// SIMATIC S7-200 project (STEP 7-Micro/WIN), CPU 222 REL 02.01

ORGANIZATION_BLOCK MAIN:OB1
TITLE=
BEGIN
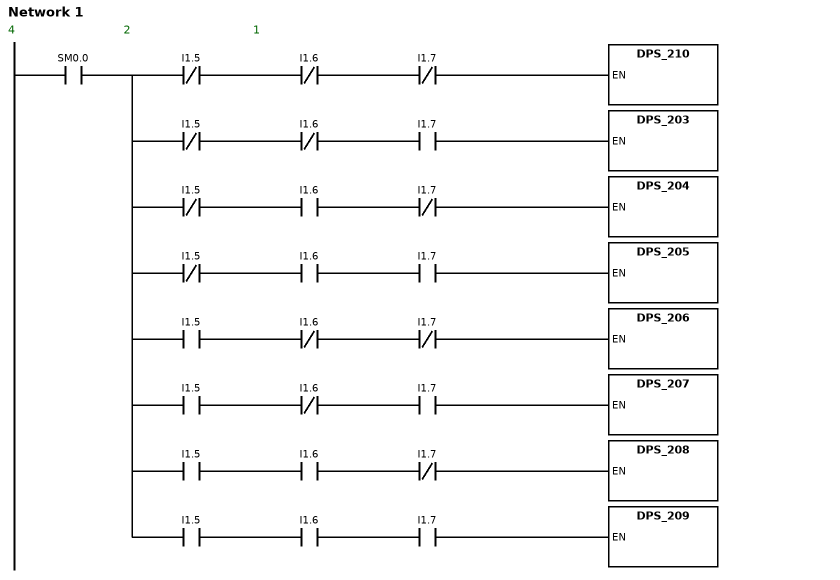
Network 1
//                                            4                               2                                   1
LD     SM0.0
LPS
AN     I1.5
AN     I1.6
AN     I1.7
CALL   DPS_210:SBR2
LRD
AN     I1.5
AN     I1.6
A      I1.7
CALL   DPS_203:SBR3
LRD
AN     I1.5
A      I1.6
AN     I1.7
CALL   DPS_204:SBR4
LRD
AN     I1.5
A      I1.6
A      I1.7
CALL   DPS_205:SBR7
LRD
A      I1.5
AN     I1.6
AN     I1.7
CALL   DPS_206:SBR8
LRD
A      I1.5
AN     I1.6
A      I1.7
CALL   DPS_207:SBR9
LRD
A      I1.5
A      I1.6
AN     I1.7
CALL   DPS_208:SBR14
LPP
A      I1.5
A      I1.6
A      I1.7
CALL   DPS_209:SBR15
END_ORGANIZATION_BLOCK

SUBROUTINE_BLOCK SCALA:SBR0
TITLE=COMMENTI SUL SOTTOPROGRAMMA
VAR_INPUT
x:WORD;	// LW0 
x1:REAL;	// LD2 
x2:REAL;	// LD6 
y1:REAL;	// LD10 
y2:REAL;	// LD14 
END_VAR
VAR_OUTPUT
y:REAL;	// LD18 
END_VAR
BEGIN
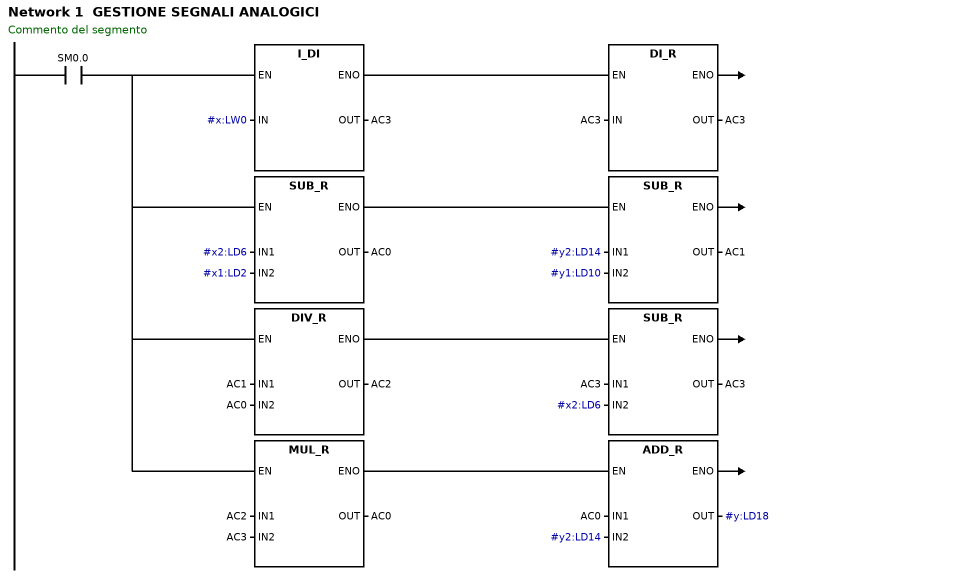
Network 1 // GESTIONE SEGNALI ANALOGICI
// Commento del segmento
LD     SM0.0
LPS
ITD    #x:LW0, AC3
AENO
DTR    AC3, AC3
LRD
MOVR   #x2:LD6, AC0
AENO
-R     #x1:LD2, AC0
AENO
MOVR   #y2:LD14, AC1
-R     #y1:LD10, AC1
LRD
MOVR   AC1, AC2
AENO
/R     AC0, AC2
AENO
-R     #x2:LD6, AC3
LPP
MOVR   AC2, AC0
AENO
*R     AC3, AC0
AENO
MOVR   AC0, #y:LD18
+R     #y2:LD14, #y:LD18
Network 2 // Titolo del segmento
// Commento del segmento
END_SUBROUTINE_BLOCK

SUBROUTINE_BLOCK MISURE:SBR1
TITLE=SCALA GLI INGRESSI ANALOGICI DA 0-100
BEGIN
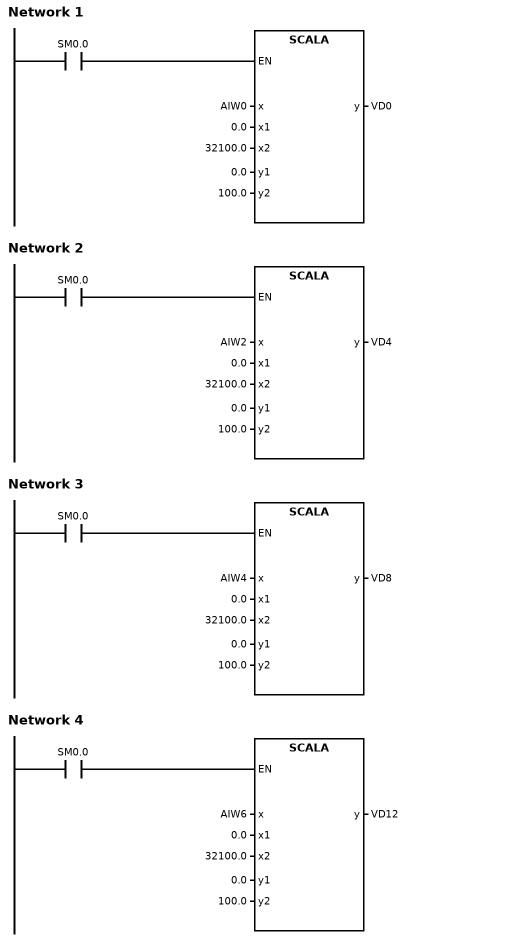
Network 1
LD     SM0.0
CALL   SCALA:SBR0, AIW0, 0.0, 32100.0, 0.0, 100.0, VD0
Network 2
LD     SM0.0
CALL   SCALA:SBR0, AIW2, 0.0, 32100.0, 0.0, 100.0, VD4
Network 3
LD     SM0.0
CALL   SCALA:SBR0, AIW4, 0.0, 32100.0, 0.0, 100.0, VD8
Network 4
LD     SM0.0
CALL   SCALA:SBR0, AIW6, 0.0, 32100.0, 0.0, 100.0, VD12
Network 5 // Titolo del segmento
// Commento del segmento
END_SUBROUTINE_BLOCK

SUBROUTINE_BLOCK DPS_210:SBR2
TITLE=DPS 210 IMPIANTO DI RISCALDAMENTO
BEGIN
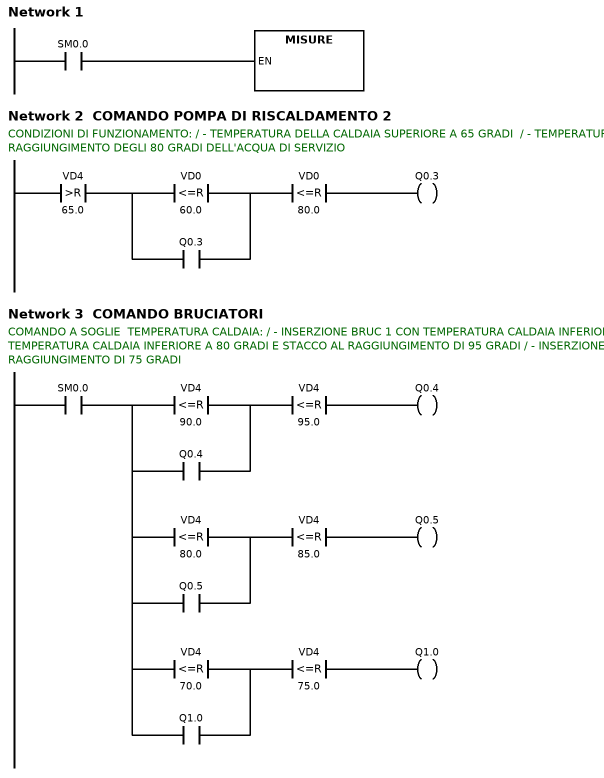
Network 1
LD     SM0.0
CALL   MISURE:SBR1
Network 2 // COMANDO POMPA DI RISCALDAMENTO 2
// CONDIZIONI DI FUNZIONAMENTO:
// - TEMPERATURA DELLA CALDAIA SUPERIORE A 65 GRADI 
// - TEMPERATURA DI SERVIZIO INFERIORE A 60 GRADI
// PARTE LA POMPA DI CIRCOLAZIONE 2 FINO AL RAGGIUNGIMENTO DEGLI 80 GRADI DELL'ACQUA DI SERVIZIO
LDR>   VD4, 65.0
LDR<=  VD0, 60.0
O      Q0.3
ALD
AR<=   VD0, 80.0
=      Q0.3
Network 3 // COMANDO BRUCIATORI
// COMANDO A SOGLIE  TEMPERATURA CALDAIA:
// - INSERZIONE BRUC 1 CON TEMPERATURA CALDAIA INFERIORE A 90 GRADI E STACCO AL RAGGIUNGIMENTO DI 95 GRADI
// - INSERZIONE BRUC 2 CON TEMPERATURA CALDAIA INFERIORE A 80 GRADI E STACCO AL RAGGIUNGIMENTO DI 95 GRADI
// - INSERZIONE BRUC 3 CON TEMPERATURA CALDAIA INFERIORE A 70 GRADI E STACCO AL RAGGIUNGIMENTO DI 75 GRADI
LD     SM0.0
LPS
LDR<=  VD4, 90.0
O      Q0.4
ALD
AR<=   VD4, 95.0
=      Q0.4
LRD
LDR<=  VD4, 80.0
O      Q0.5
ALD
AR<=   VD4, 85.0
=      Q0.5
LPP
LDR<=  VD4, 70.0
O      Q1.0
ALD
AR<=   VD4, 75.0
=      Q1.0
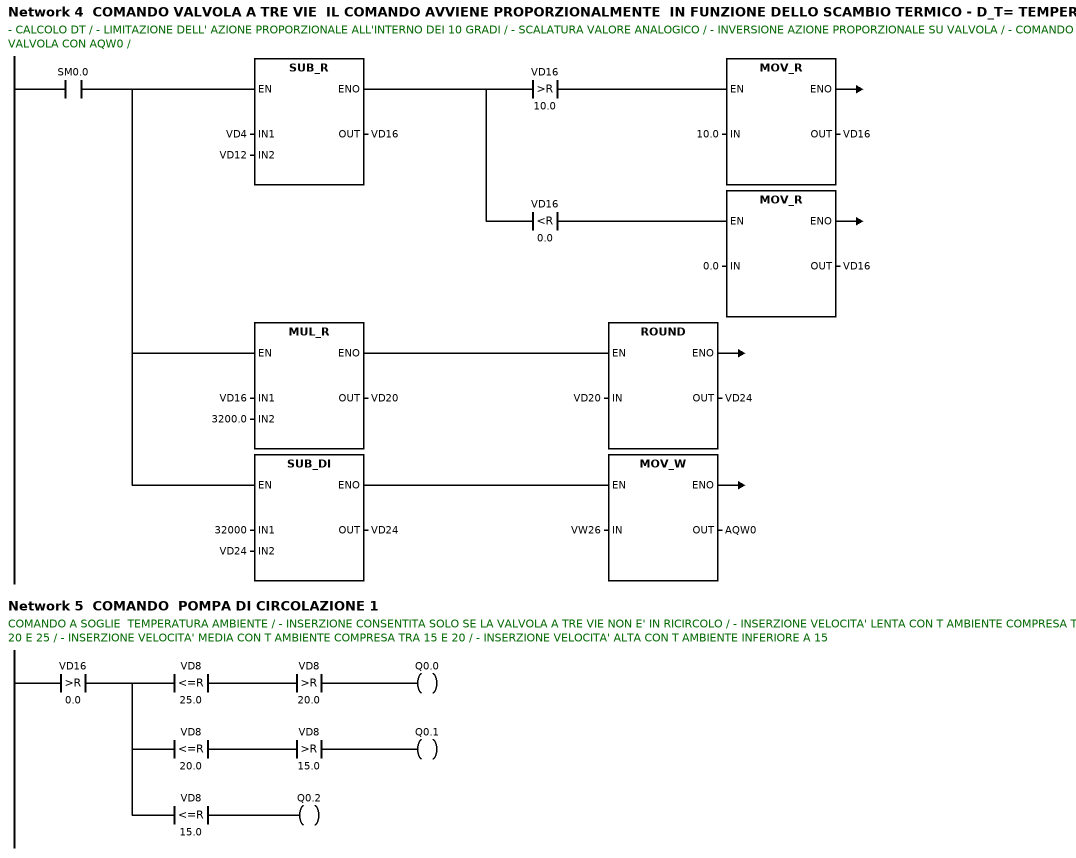
Network 4 // COMANDO VALVOLA A TRE VIE 
IL COMANDO AVVIENE PROPORZIONALMENTE  IN FUNZIONE DELLO SCAMBIO TERMICO
- D_T= TEMPERATURA CALDAIA - TEMPERATURA RITORNO
- D_T =0 VALVOLA TRE VIE IN RICIRCOLO
- D_T= 10 VALVOLA TRE VIE IN PIENA MANDATA
// - CALCOLO DT
// - LIMITAZIONE DELL' AZIONE PROPORZIONALE ALL'INTERNO DEI 10 GRADI
// - SCALATURA VALORE ANALOGICO
// - INVERSIONE AZIONE PROPORZIONALE SU VALVOLA
// - COMANDO VALVOLA CON AQW0
// 
LD     SM0.0
LPS
MOVR   VD4, VD16
AENO
-R     VD12, VD16
AENO
LPS
AR>    VD16, 10.0
MOVR   10.0, VD16
LPP
AR<    VD16, 0.0
MOVR   0.0, VD16
LPP
LPS
MOVR   VD16, VD20
AENO
*R     3200.0, VD20
AENO
ROUND  VD20, VD24
LPP
INVD   VD24
AENO
INCD   VD24
AENO
+D     32000, VD24
AENO
MOVW   VW26, AQW0
Network 5 // COMANDO  POMPA DI CIRCOLAZIONE 1
// COMANDO A SOGLIE  TEMPERATURA AMBIENTE
// - INSERZIONE CONSENTITA SOLO SE LA VALVOLA A TRE VIE NON E' IN RICIRCOLO
// - INSERZIONE VELOCITA' LENTA CON T AMBIENTE COMPRESA TRA 20 E 25
// - INSERZIONE VELOCITA' MEDIA CON T AMBIENTE COMPRESA TRA 15 E 20
// - INSERZIONE VELOCITA' ALTA CON T AMBIENTE INFERIORE A 15
LDR>   VD16, 0.0
LPS
AR<=   VD8, 25.0
AR>    VD8, 20.0
=      Q0.0
LRD
AR<=   VD8, 20.0
AR>    VD8, 15.0
=      Q0.1
LPP
AR<=   VD8, 15.0
=      Q0.2
Network 9 // Titolo del segmento
// Commento del segmento
END_SUBROUTINE_BLOCK

SUBROUTINE_BLOCK DPS_203:SBR3
TITLE=DPS 203 MONTACARICHI
BEGIN
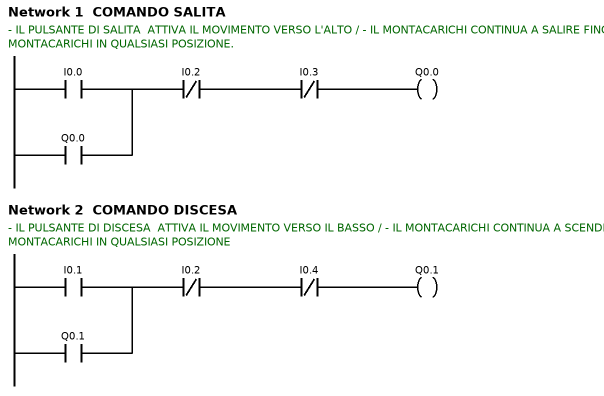
Network 1 // COMANDO SALITA 
// - IL PULSANTE DI SALITA  ATTIVA IL MOVIMENTO VERSO L'ALTO
// - IL MONTACARICHI CONTINUA A SALIRE FINO AL' INTERVENTO DEL FC_SUP
// - IL PULSANTE DI STOP ARRESTA LA SALITA DEL  MONTACARICHI IN QUALSIASI POSIZIONE.
LD     I0.0
O      Q0.0
AN     I0.2
AN     I0.3
=      Q0.0
Network 2 // COMANDO DISCESA
// - IL PULSANTE DI DISCESA  ATTIVA IL MOVIMENTO VERSO IL BASSO
// - IL MONTACARICHI CONTINUA A SCENDERE FINO AL' INTERVENTO DEL FC_INF
// - IL PULSANTE DI STOP ARRESTA LA DISCESA  DEL  MONTACARICHI IN QUALSIASI POSIZIONE
LD     I0.1
O      Q0.1
AN     I0.2
AN     I0.4
=      Q0.1
Network 28 // Titolo del segmento
// Commento del segmento
END_SUBROUTINE_BLOCK

SUBROUTINE_BLOCK DPS_204:SBR4
TITLE=DPS 204 DISTRIBUTORE BEVANDE
BEGIN
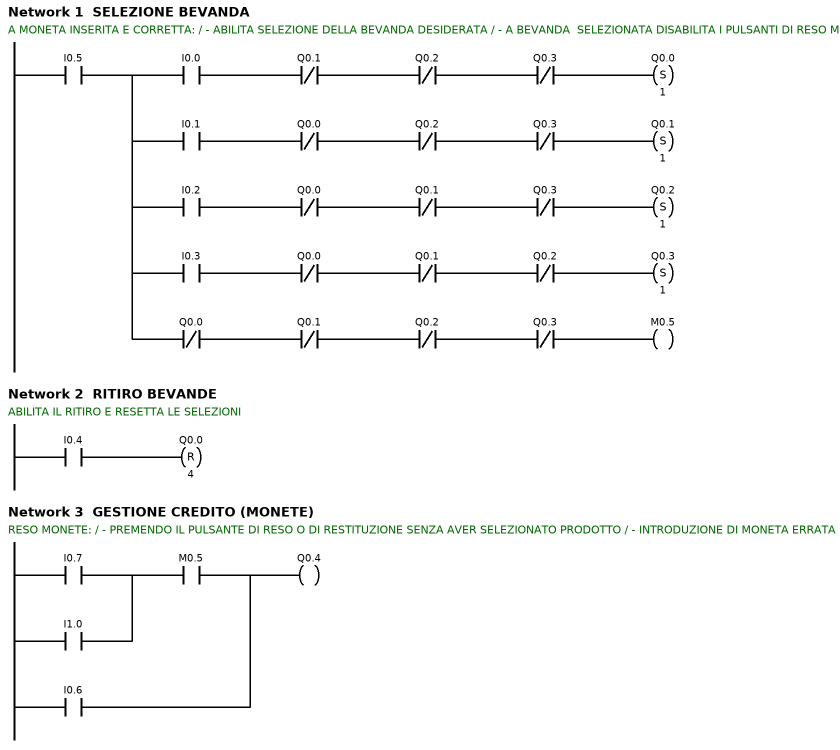
Network 1 // SELEZIONE BEVANDA
// A MONETA INSERITA E CORRETTA:
// - ABILITA SELEZIONE DELLA BEVANDA DESIDERATA
// - A BEVANDA  SELEZIONATA DISABILITA I PULSANTI DI RESO MONETA E RESTITUZIONE MONETA
// 
LD     I0.5
LPS
A      I0.0
AN     Q0.1
AN     Q0.2
AN     Q0.3
S      Q0.0, 1
LRD
A      I0.1
AN     Q0.0
AN     Q0.2
AN     Q0.3
S      Q0.1, 1
LRD
A      I0.2
AN     Q0.0
AN     Q0.1
AN     Q0.3
S      Q0.2, 1
LRD
A      I0.3
AN     Q0.0
AN     Q0.1
AN     Q0.2
S      Q0.3, 1
LPP
AN     Q0.0
AN     Q0.1
AN     Q0.2
AN     Q0.3
=      M0.5
Network 2 // RITIRO BEVANDE
// ABILITA IL RITIRO E RESETTA LE SELEZIONI
LD     I0.4
R      Q0.0, 4
Network 3 // GESTIONE CREDITO (MONETE)
// RESO MONETE:
// - PREMENDO IL PULSANTE DI RESO O DI RESTITUZIONE SENZA AVER SELEZIONATO PRODOTTO
// - INTRODUZIONE DI MONETA ERRATA
LD     I0.7
O      I1.0
A      M0.5
O      I0.6
=      Q0.4
Network 4
// MEND
Network 5 // Titolo del segmento
// Commento del segmento
END_SUBROUTINE_BLOCK

SUBROUTINE_BLOCK AUT_205:SBR5
TITLE=
BEGIN
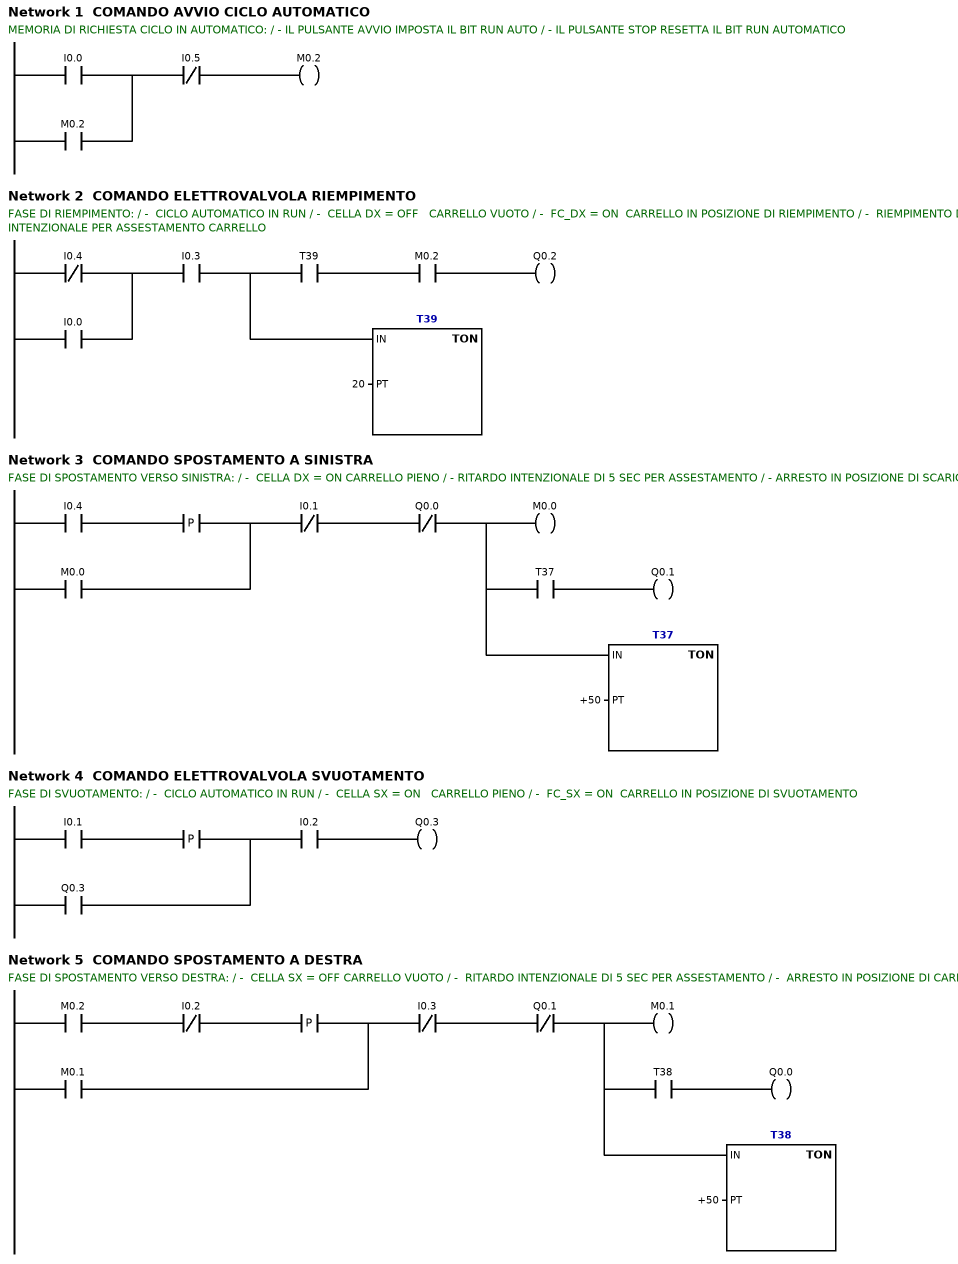
Network 1 // COMANDO AVVIO CICLO AUTOMATICO
// MEMORIA DI RICHIESTA CICLO IN AUTOMATICO:
// - IL PULSANTE AVVIO IMPOSTA IL BIT RUN AUTO
// - IL PULSANTE STOP RESETTA IL BIT RUN AUTOMATICO
LD     I0.0
O      M0.2
AN     I0.5
=      M0.2
Network 2 // COMANDO ELETTROVALVOLA RIEMPIMENTO
// FASE DI RIEMPIMENTO:
// -  CICLO AUTOMATICO IN RUN
// -  CELLA DX = OFF   CARRELLO VUOTO
// -  FC_DX = ON  CARRELLO IN POSIZIONE DI RIEMPIMENTO
// -  RIEMPIMENTO DOPO RITARDO INTENZIONALE PER ASSESTAMENTO CARRELLO
LDN    I0.4
O      I0.0
A      I0.3
LPS
A      T39
A      M0.2
=      Q0.2
LPP
TON    T39, 20
Network 3 // COMANDO SPOSTAMENTO A SINISTRA
// FASE DI SPOSTAMENTO VERSO SINISTRA:
// -  CELLA DX = ON CARRELLO PIENO
// - RITARDO INTENZIONALE DI 5 SEC PER ASSESTAMENTO
// - ARRESTO IN POSIZIONE DI SCARICO FC_SX = ON
LD     I0.4
EU
O      M0.0
AN     I0.1
AN     Q0.0
LPS
=      M0.0
A      T37
=      Q0.1
LPP
TON    T37, +50
Network 4 // COMANDO ELETTROVALVOLA SVUOTAMENTO
// FASE DI SVUOTAMENTO:
// -  CICLO AUTOMATICO IN RUN
// -  CELLA SX = ON   CARRELLO PIENO
// -  FC_SX = ON  CARRELLO IN POSIZIONE DI SVUOTAMENTO
LD     I0.1
EU
O      Q0.3
A      I0.2
=      Q0.3
Network 5 // COMANDO SPOSTAMENTO A DESTRA
// FASE DI SPOSTAMENTO VERSO DESTRA:
// -  CELLA SX = OFF CARRELLO VUOTO
// -  RITARDO INTENZIONALE DI 5 SEC PER ASSESTAMENTO
// -  ARRESTO IN POSIZIONE DI CARICO FC_DX = ON
LD     M0.2
AN     I0.2
EU
O      M0.1
AN     I0.3
AN     Q0.1
LPS
=      M0.1
A      T38
=      Q0.0
LPP
TON    T38, +50
END_SUBROUTINE_BLOCK

SUBROUTINE_BLOCK MAN_205:SBR6
TITLE=
BEGIN
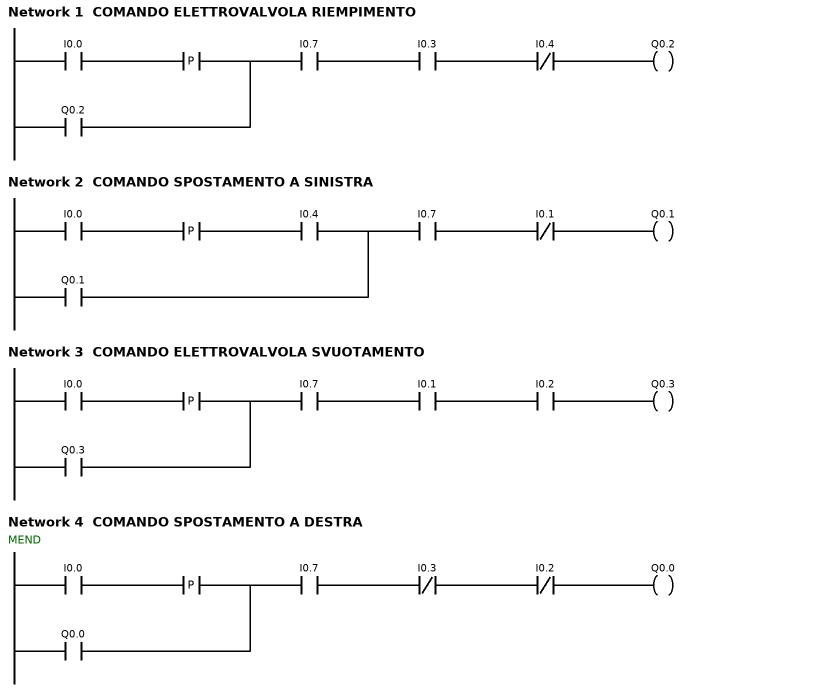
Network 1 // COMANDO ELETTROVALVOLA RIEMPIMENTO
LD     I0.0
EU
O      Q0.2
A      I0.7
A      I0.3
AN     I0.4
=      Q0.2
Network 2 // COMANDO SPOSTAMENTO A SINISTRA
LD     I0.0
EU
A      I0.4
O      Q0.1
A      I0.7
AN     I0.1
=      Q0.1
Network 3 // COMANDO ELETTROVALVOLA SVUOTAMENTO
LD     I0.0
EU
O      Q0.3
A      I0.7
A      I0.1
A      I0.2
=      Q0.3
Network 4 // COMANDO SPOSTAMENTO A DESTRA
// MEND
LD     I0.0
EU
O      Q0.0
A      I0.7
AN     I0.3
AN     I0.2
=      Q0.0
Network 5 // Ti
// Commento del segmento
END_SUBROUTINE_BLOCK

SUBROUTINE_BLOCK DPS_205:SBR7
TITLE=DPS 205 TRASPORTO MATERIALE SFUSO
// 
BEGIN
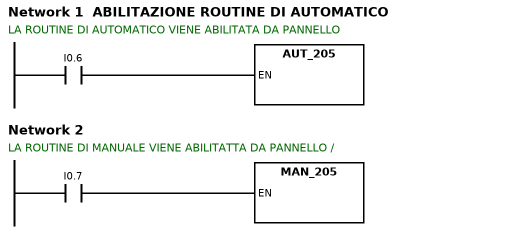
Network 1 // ABILITAZIONE ROUTINE DI AUTOMATICO
// LA ROUTINE DI AUTOMATICO VIENE ABILITATA DA PANNELLO
LD     I0.6
CALL   AUT_205:SBR5
Network 2
// LA ROUTINE DI MANUALE VIENE ABILITATTA DA PANNELLO
// 
LD     I0.7
CALL   MAN_205:SBR6
Network 26 // Titolo del segmento
// Commento del segmento
END_SUBROUTINE_BLOCK

SUBROUTINE_BLOCK DPS_206:SBR8
TITLE=DPS 206 DISPOSITIVO DI IMBOTTIGLIAMENTO
BEGIN
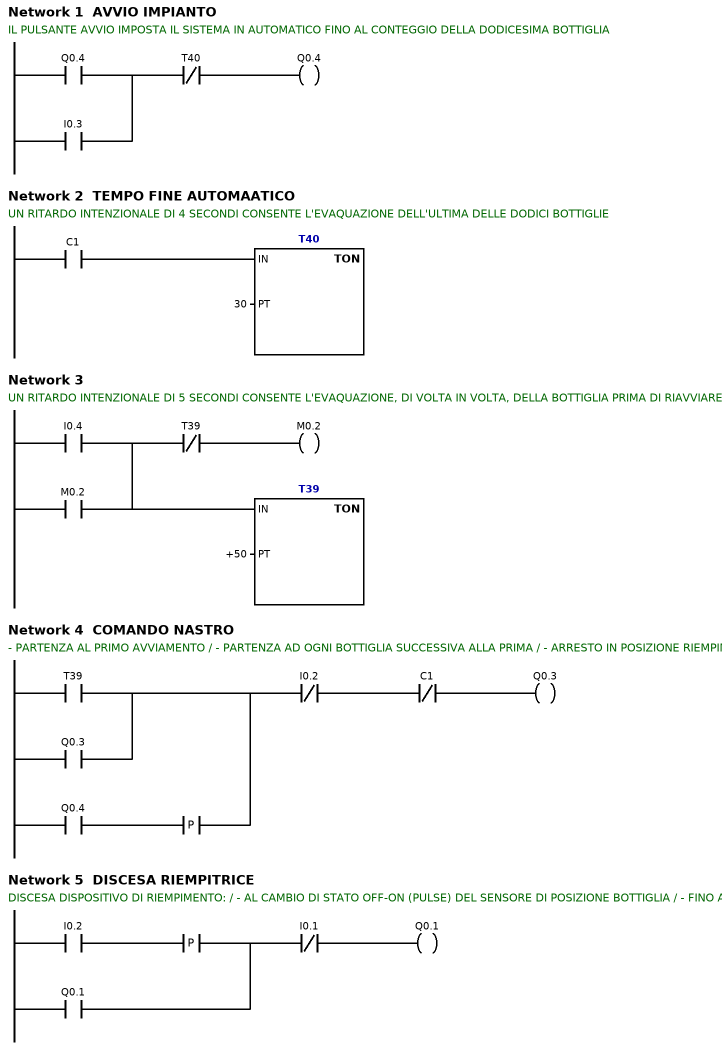
Network 1 // AVVIO IMPIANTO
// IL PULSANTE AVVIO IMPOSTA IL SISTEMA IN AUTOMATICO FINO AL CONTEGGIO DELLA DODICESIMA BOTTIGLIA
LD     Q0.4
O      I0.3
AN     T40
=      Q0.4
Network 2 // TEMPO FINE AUTOMAATICO
// UN RITARDO INTENZIONALE DI 4 SECONDI CONSENTE L'EVAQUAZIONE DELL'ULTIMA DELLE DODICI BOTTIGLIE
LD     C1
TON    T40, 30
Network 3
// UN RITARDO INTENZIONALE DI 5 SECONDI CONSENTE L'EVAQUAZIONE, DI VOLTA IN VOLTA, DELLA BOTTIGLIA PRIMA DI RIAVVIARE IL NASTRO
LD     I0.4
O      M0.2
LPS
AN     T39
=      M0.2
LPP
TON    T39, +50
Network 4 // COMANDO NASTRO
// - PARTENZA AL PRIMO AVVIAMENTO
// - PARTENZA AD OGNI BOTTIGLIA SUCCESSIVA ALLA PRIMA
// - ARRESTO IN POSIZIONE RIEMPIMENTO
// - ARRESTO A CASSA PIENA
LD     T39
O      Q0.3
LD     Q0.4
EU
OLD
AN     I0.2
AN     C1
=      Q0.3
Network 5 // DISCESA RIEMPITRICE
// DISCESA DISPOSITIVO DI RIEMPIMENTO:
// - AL CAMBIO DI STATO OFF-ON (PULSE) DEL SENSORE DI POSIZIONE BOTTIGLIA
// - FINO AD IMPEGNARE IL FINECORSA INFERIORE FC_INF=ON
// 
LD     I0.2
EU
O      Q0.1
AN     I0.1
=      Q0.1
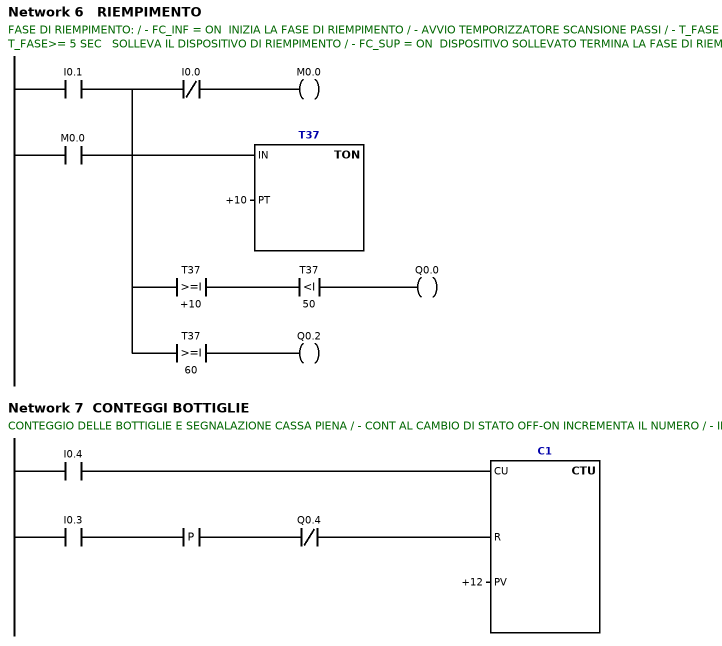
Network 6 //  RIEMPIMENTO
// FASE DI RIEMPIMENTO:
// - FC_INF = ON  INIZIA LA FASE DI RIEMPIMENTO
// - AVVIO TEMPORIZZATORE SCANSIONE PASSI
// - T_FASE >= 1 SEC  FINO A T_FASE < 4 SEC TIENE APERTO IL DOSATORE 
// - T_FASE>= 5 SEC   SOLLEVA IL DISPOSITIVO DI RIEMPIMENTO
// - FC_SUP = ON  DISPOSITIVO SOLLEVATO TERMINA LA FASE DI RIEMPIMENTO.
// 
LD     I0.1
O      M0.0
LPS
AN     I0.0
=      M0.0
LRD
TON    T37, +10
LRD
AW>=   T37, +10
AW<    T37, 50
=      Q0.0
LPP
AW>=   T37, 60
=      Q0.2
Network 7 // CONTEGGI BOTTIGLIE
// CONTEGGIO DELLE BOTTIGLIE E SEGNALAZIONE CASSA PIENA
// - CONT AL CAMBIO DI STATO OFF-ON INCREMENTA IL NUMERO
// - IL CONTEGGIO SI AZZERA AL RIAVVIO
LD     I0.4
LD     I0.3
EU
AN     Q0.4
CTU    C1, +12
Network 26 // Titolo del segmento
// Commento del segmento
END_SUBROUTINE_BLOCK

SUBROUTINE_BLOCK DPS_207:SBR9
TITLE=DPS 207 NASTRO TRASPORTATORE
BEGIN
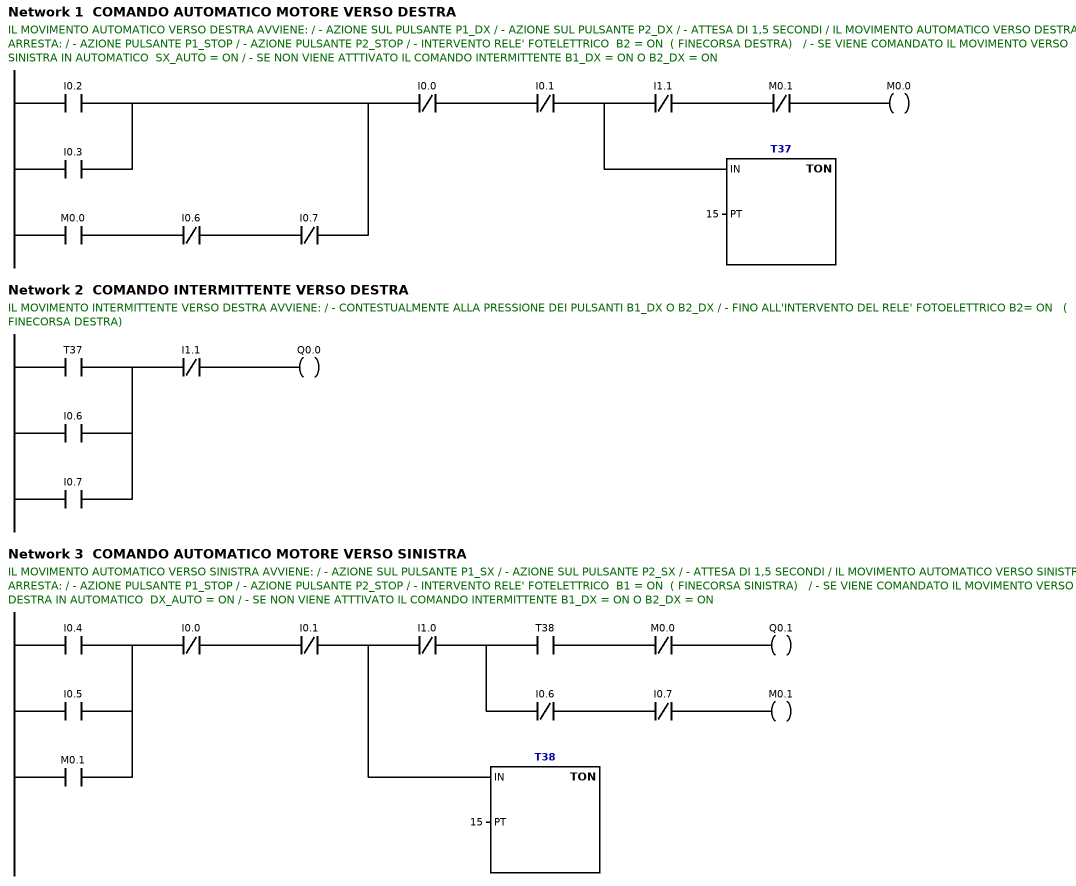
Network 1 // COMANDO AUTOMATICO MOTORE VERSO DESTRA
// IL MOVIMENTO AUTOMATICO VERSO DESTRA AVVIENE:
// - AZIONE SUL PULSANTE P1_DX
// - AZIONE SUL PULSANTE P2_DX
// - ATTESA DI 1,5 SECONDI
// IL MOVIMENTO AUTOMATICO VERSO DESTRA SI ARRESTA:
// - AZIONE PULSANTE P1_STOP
// - AZIONE PULSANTE P2_STOP
// - INTERVENTO RELE' FOTELETTRICO  B2 = ON  ( FINECORSA DESTRA)  
// - SE VIENE COMANDATO IL MOVIMENTO VERSO SINISTRA IN AUTOMATICO  SX_AUTO = ON
// - SE NON VIENE ATTTIVATO IL COMANDO INTERMITTENTE B1_DX = ON O B2_DX = ON
LD     I0.2
O      I0.3
LD     M0.0
AN     I0.6
AN     I0.7
OLD
AN     I0.0
AN     I0.1
LPS
AN     I1.1
AN     M0.1
=      M0.0
LPP
TON    T37, 15
Network 2 // COMANDO INTERMITTENTE VERSO DESTRA
// IL MOVIMENTO INTERMITTENTE VERSO DESTRA AVVIENE:
// - CONTESTUALMENTE ALLA PRESSIONE DEI PULSANTI B1_DX O B2_DX
// - FINO ALL'INTERVENTO DEL RELE' FOTOELETTRICO B2= ON   ( FINECORSA DESTRA)  
LD     T37
O      I0.6
O      I0.7
AN     I1.1
=      Q0.0
Network 3 // COMANDO AUTOMATICO MOTORE VERSO SINISTRA
// IL MOVIMENTO AUTOMATICO VERSO SINISTRA AVVIENE:
// - AZIONE SUL PULSANTE P1_SX
// - AZIONE SUL PULSANTE P2_SX
// - ATTESA DI 1,5 SECONDI
// IL MOVIMENTO AUTOMATICO VERSO SINISTRA SI ARRESTA:
// - AZIONE PULSANTE P1_STOP
// - AZIONE PULSANTE P2_STOP
// - INTERVENTO RELE' FOTELETTRICO  B1 = ON  ( FINECORSA SINISTRA)  
// - SE VIENE COMANDATO IL MOVIMENTO VERSO DESTRA IN AUTOMATICO  DX_AUTO = ON
// - SE NON VIENE ATTTIVATO IL COMANDO INTERMITTENTE B1_DX = ON O B2_DX = ON
LD     I0.4
O      I0.5
O      M0.1
AN     I0.0
AN     I0.1
LPS
AN     I1.0
LPS
A      T38
AN     M0.0
=      Q0.1
LPP
AN     I0.6
AN     I0.7
=      M0.1
LPP
TON    T38, 15
Network 7 // Titolo del segmento
// Commento del segmento
END_SUBROUTINE_BLOCK

SUBROUTINE_BLOCK SEM_208:SBR10
TITLE=
BEGIN
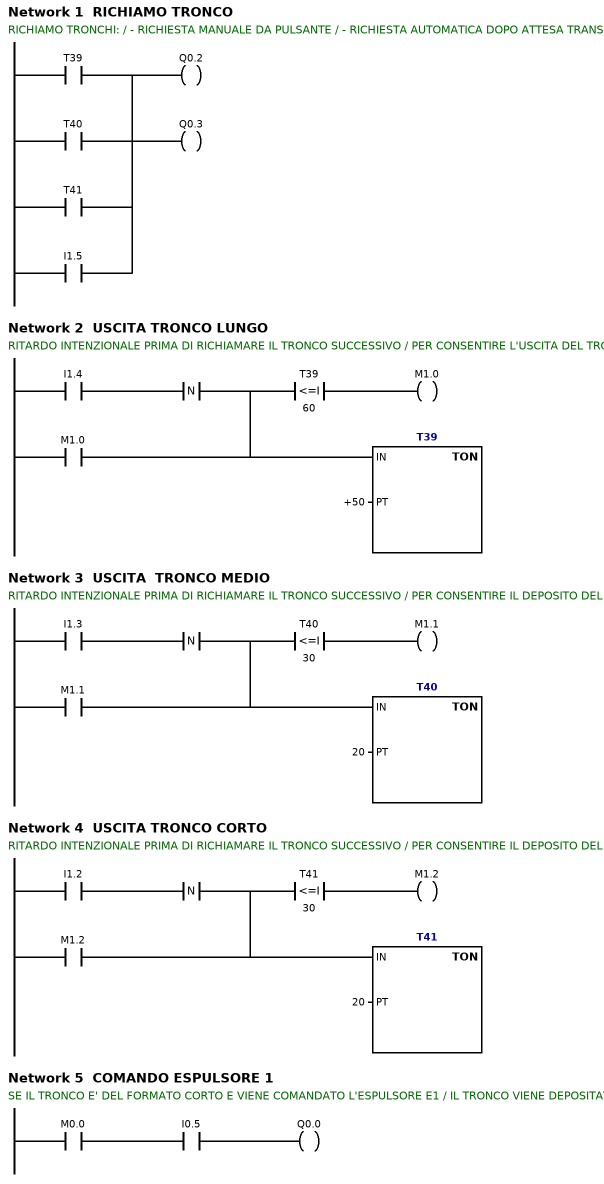
Network 1 // RICHIAMO TRONCO
// RICHIAMO TRONCHI:
// - RICHIESTA MANUALE DA PULSANTE
// - RICHIESTA AUTOMATICA DOPO ATTESA TRANSITO COMPLETO DEL TRONCO PRECEDENTE
LD     T39
O      T40
O      T41
O      I1.5
=      Q0.2
=      Q0.3
Network 2 // USCITA TRONCO LUNGO
// RITARDO INTENZIONALE PRIMA DI RICHIAMARE IL TRONCO SUCCESSIVO
// PER CONSENTIRE L'USCITA DEL TRONCO LUNGO
LD     I1.4
ED
O      M1.0
LPS
AW<=   T39, 60
=      M1.0
LPP
TON    T39, +50
Network 3 // USCITA  TRONCO MEDIO
// RITARDO INTENZIONALE PRIMA DI RICHIAMARE IL TRONCO SUCCESSIVO
// PER CONSENTIRE IL DEPOSITO DEL TRONCO MEDIO NEL BOX 2
LD     I1.3
ED
O      M1.1
LPS
AW<=   T40, 30
=      M1.1
LPP
TON    T40, 20
Network 4 // USCITA TRONCO CORTO
// RITARDO INTENZIONALE PRIMA DI RICHIAMARE IL TRONCO SUCCESSIVO
// PER CONSENTIRE IL DEPOSITO DEL TRONCO CORTO NEL BOX 1
LD     I1.2
ED
O      M1.2
LPS
AW<=   T41, 30
=      M1.2
LPP
TON    T41, 20
Network 5 // COMANDO ESPULSORE 1
// SE IL TRONCO E' DEL FORMATO CORTO E VIENE COMANDATO L'ESPULSORE E1
// IL TRONCO VIENE DEPOSITATO NEL BOX 1
LD     M0.0
A      I0.5
=      Q0.0
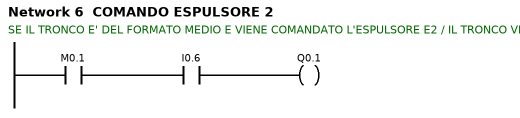
Network 6 // COMANDO ESPULSORE 2
// SE IL TRONCO E' DEL FORMATO MEDIO E VIENE COMANDATO L'ESPULSORE E2
// IL TRONCO VIENE DEPOSITATO NEL BOX 2
LD     M0.1
A      I0.6
=      Q0.1
Network 13 // Titolo del segmento
// Commento del segmento
END_SUBROUTINE_BLOCK

SUBROUTINE_BLOCK AUT_208:SBR11
TITLE=
BEGIN
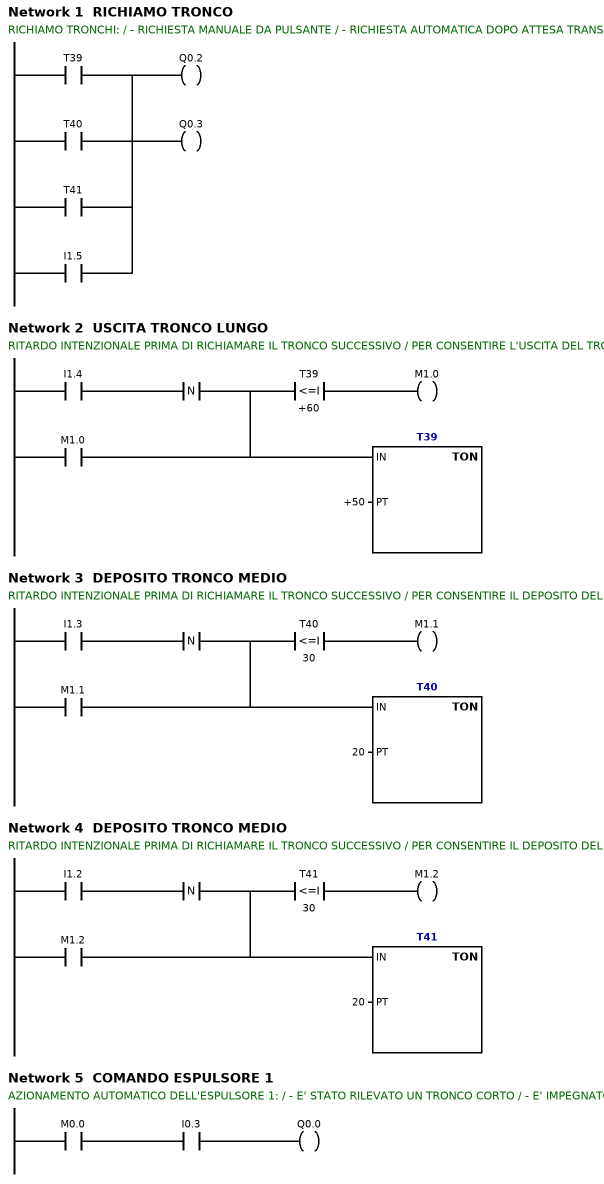
Network 1 // RICHIAMO TRONCO
// RICHIAMO TRONCHI:
// - RICHIESTA MANUALE DA PULSANTE
// - RICHIESTA AUTOMATICA DOPO ATTESA TRANSITO COMPLETO DEL TRONCO PRECEDENTE
LD     T39
O      T40
O      T41
O      I1.5
=      Q0.2
=      Q0.3
Network 2 // USCITA TRONCO LUNGO
// RITARDO INTENZIONALE PRIMA DI RICHIAMARE IL TRONCO SUCCESSIVO
// PER CONSENTIRE L'USCITA DEL TRONCO LUNGO
LD     I1.4
ED
O      M1.0
LPS
AW<=   T39, +60
=      M1.0
LPP
TON    T39, +50
Network 3 // DEPOSITO TRONCO MEDIO
// RITARDO INTENZIONALE PRIMA DI RICHIAMARE IL TRONCO SUCCESSIVO
// PER CONSENTIRE IL DEPOSITO DEL TRONCO MEDIO NEL BOX 2
LD     I1.3
ED
O      M1.1
LPS
AW<=   T40, 30
=      M1.1
LPP
TON    T40, 20
Network 4 // DEPOSITO TRONCO MEDIO
// RITARDO INTENZIONALE PRIMA DI RICHIAMARE IL TRONCO SUCCESSIVO
// PER CONSENTIRE IL DEPOSITO DEL TRONCO CORTO NEL BOX 1
LD     I1.2
ED
O      M1.2
LPS
AW<=   T41, 30
=      M1.2
LPP
TON    T41, 20
Network 5 // COMANDO ESPULSORE 1
// AZIONAMENTO AUTOMATICO DELL'ESPULSORE 1:
// - E' STATO RILEVATO UN TRONCO CORTO
// - E' IMPEGNATO IL TRASCINATORE B7
LD     M0.0
A      I0.3
=      Q0.0
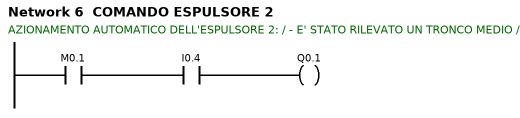
Network 6 // COMANDO ESPULSORE 2
// AZIONAMENTO AUTOMATICO DELL'ESPULSORE 2:
// - E' STATO RILEVATO UN TRONCO MEDIO
// - E' IMPEGNATO IL TRASCINATORE B8
LD     M0.1
A      I0.4
=      Q0.1
END_SUBROUTINE_BLOCK

SUBROUTINE_BLOCK SELEZIONE:SBR12
TITLE=
BEGIN
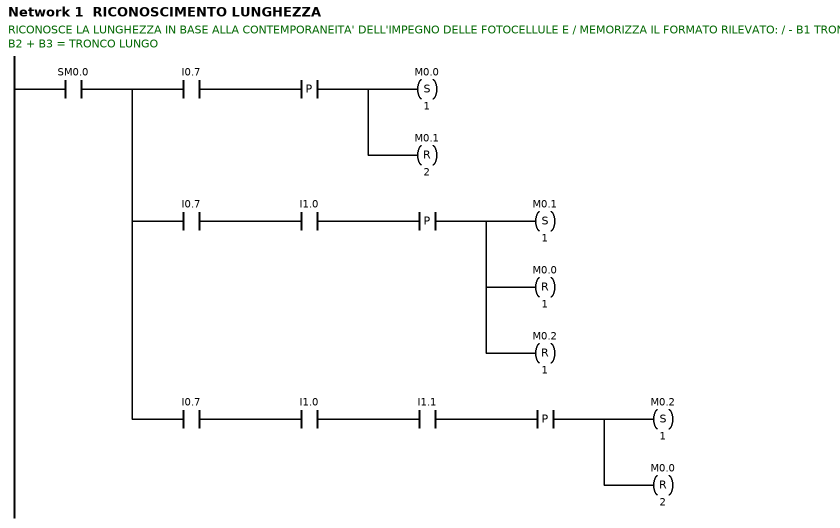
Network 1 // RICONOSCIMENTO LUNGHEZZA
// RICONOSCE LA LUNGHEZZA IN BASE ALLA CONTEMPORANEITA' DELL'IMPEGNO DELLE FOTOCELLULE E
// MEMORIZZA IL FORMATO RILEVATO:
// - B1 TRONCO CORTO
// - B1+ B2 TRONCO MEDIO
// - B1 + B2 + B3 = TRONCO LUNGO
LD     SM0.0
LPS
A      I0.7
EU
S      M0.0, 1
R      M0.1, 2
LRD
A      I0.7
A      I1.0
EU
S      M0.1, 1
R      M0.0, 1
R      M0.2, 1
LPP
A      I0.7
A      I1.0
A      I1.1
EU
S      M0.2, 1
R      M0.0, 2
Network 2 // Titolo del segmento
// Commento del segmento
END_SUBROUTINE_BLOCK

SUBROUTINE_BLOCK MAN_208:SBR13
TITLE=
BEGIN
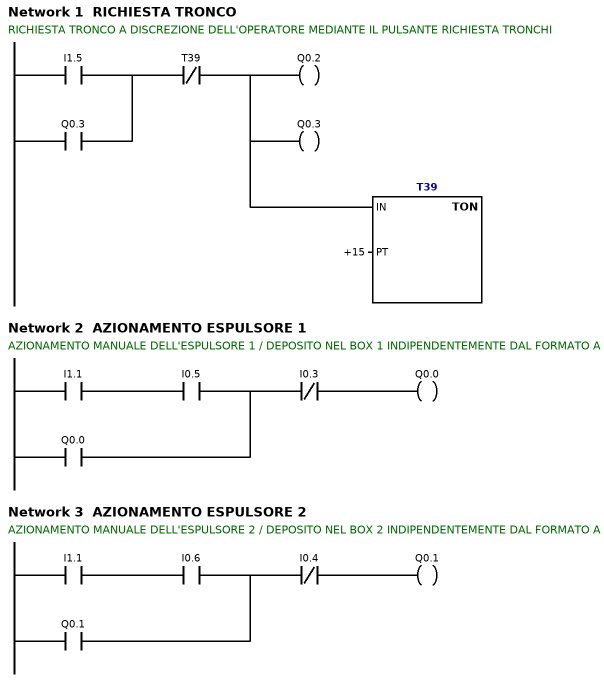
Network 1 // RICHIESTA TRONCO
// RICHIESTA TRONCO A DISCREZIONE DELL'OPERATORE MEDIANTE IL PULSANTE RICHIESTA TRONCHI
LD     I1.5
O      Q0.3
AN     T39
=      Q0.2
=      Q0.3
TON    T39, +15
Network 2 // AZIONAMENTO ESPULSORE 1
// AZIONAMENTO MANUALE DELL'ESPULSORE 1
// DEPOSITO NEL BOX 1 INDIPENDENTEMENTE DAL FORMATO A DISCREZIONE DELL'OPERATORE
LD     I1.1
A      I0.5
O      Q0.0
AN     I0.3
=      Q0.0
Network 3 // AZIONAMENTO ESPULSORE 2
// AZIONAMENTO MANUALE DELL'ESPULSORE 2
// DEPOSITO NEL BOX 2 INDIPENDENTEMENTE DAL FORMATO A DISCREZIONE DELL'OPERATORE
LD     I1.1
A      I0.6
O      Q0.1
AN     I0.4
=      Q0.1
Network 10 // Titolo del segmento
// Commento del segmento
Network 20 // Titolo del segmento
// Commento del segmento
END_SUBROUTINE_BLOCK

SUBROUTINE_BLOCK DPS_208:SBR14
TITLE=DP208 SELEZIONE LUNGHEZZE
BEGIN
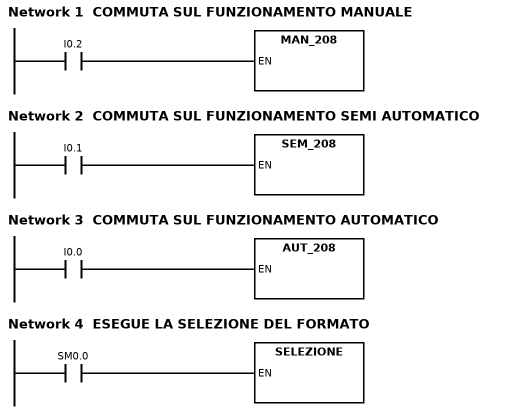
Network 1 // COMMUTA SUL FUNZIONAMENTO MANUALE
LD     I0.2
CALL   MAN_208:SBR13
Network 2 // COMMUTA SUL FUNZIONAMENTO SEMI AUTOMATICO
LD     I0.1
CALL   SEM_208:SBR10
Network 3 // COMMUTA SUL FUNZIONAMENTO AUTOMATICO
LD     I0.0
CALL   AUT_208:SBR11
Network 4 // ESEGUE LA SELEZIONE DEL FORMATO 
LD     SM0.0
CALL   SELEZIONE:SBR12
Network 26 // Titolo del segmento
// Commento del segmento
END_SUBROUTINE_BLOCK

SUBROUTINE_BLOCK DPS_209:SBR15
TITLE=SISTEMA MODULARE PER LA SIMULAZIONE DI PROCESSI INDUSTRIALI
// 
// ********** MOTORE TRIFASE***********
// 
BEGIN
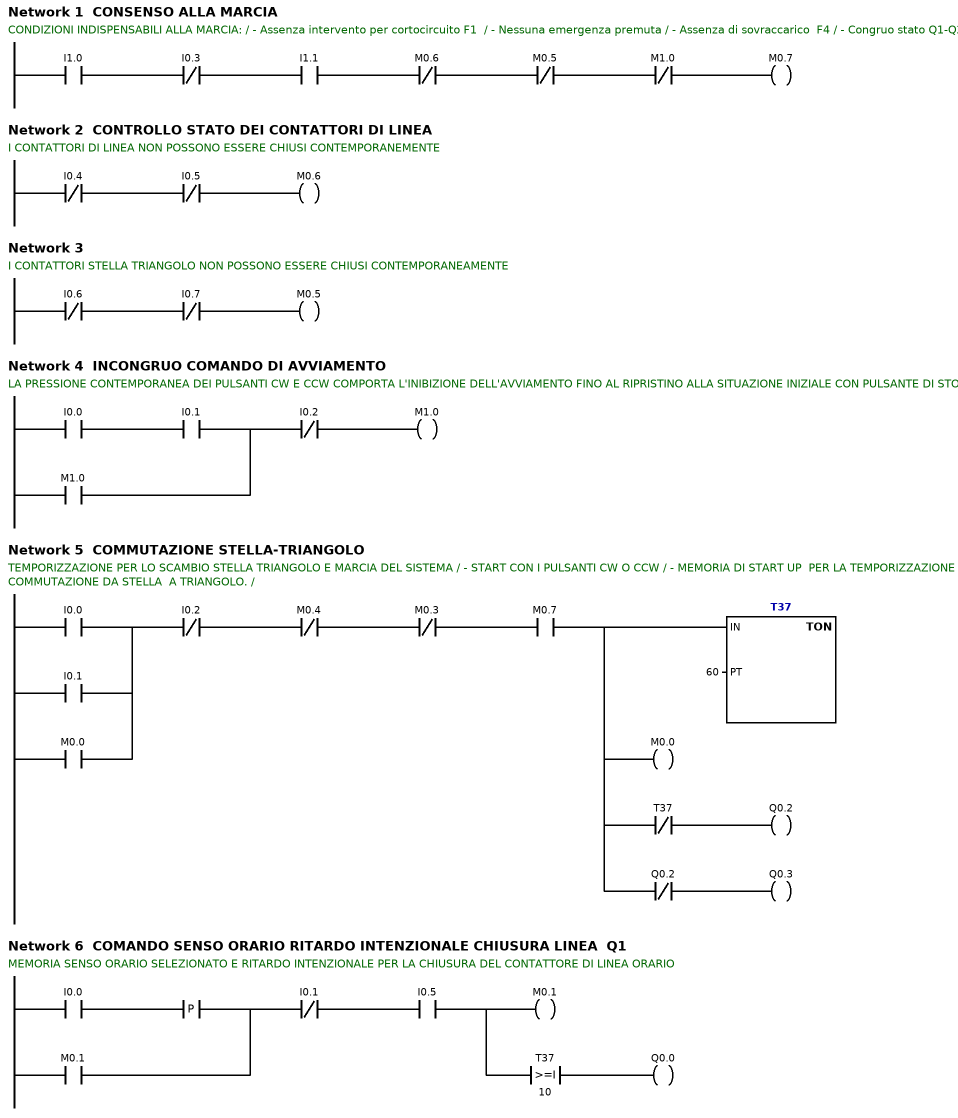
Network 1 // CONSENSO ALLA MARCIA
// CONDIZIONI INDISPENSABILI ALLA MARCIA:
// - Assenza intervento per cortocircuito F1 
// - Nessuna emergenza premuta
// - Assenza di sovraccarico  F4
// - Congruo stato Q1-Q2
// - Congruo stato Q2-Q4
// 
LD     I1.0
AN     I0.3
A      I1.1
AN     M0.6
AN     M0.5
AN     M1.0
=      M0.7
Network 2 // CONTROLLO STATO DEI CONTATTORI DI LINEA
// I CONTATTORI DI LINEA NON POSSONO ESSERE CHIUSI CONTEMPORANEMENTE
LDN    I0.4
AN     I0.5
=      M0.6
Network 3
// I CONTATTORI STELLA TRIANGOLO NON POSSONO ESSERE CHIUSI CONTEMPORANEAMENTE
LDN    I0.6
AN     I0.7
=      M0.5
Network 4 // INCONGRUO COMANDO DI AVVIAMENTO
// LA PRESSIONE CONTEMPORANEA DEI PULSANTI CW E CCW COMPORTA L'INIBIZIONE DELL'AVVIAMENTO FINO AL RIPRISTINO ALLA SITUAZIONE INIZIALE CON PULSANTE DI STOP
LD     I0.0
A      I0.1
O      M1.0
AN     I0.2
=      M1.0
Network 5 // COMMUTAZIONE STELLA-TRIANGOLO
// TEMPORIZZAZIONE PER LO SCAMBIO STELLA TRIANGOLO E MARCIA DEL SISTEMA
// - START CON I PULSANTI CW O CCW
// - MEMORIA DI START UP  PER LA TEMPORIZZAZIONE DELL'AVVIAMENTO
// - COMMUTAZIONE DA STELLA  A TRIANGOLO.
// 
LD     I0.0
O      I0.1
O      M0.0
AN     I0.2
AN     M0.4
AN     M0.3
A      M0.7
LPS
TON    T37, 60
=      M0.0
AN     T37
=      Q0.2
LPP
AN     Q0.2
=      Q0.3
Network 6 // COMANDO SENSO ORARIO RITARDO INTENZIONALE CHIUSURA LINEA  Q1
// MEMORIA SENSO ORARIO SELEZIONATO E RITARDO INTENZIONALE PER LA CHIUSURA DEL CONTATTORE DI LINEA ORARIO
LD     I0.0
EU
O      M0.1
AN     I0.1
A      I0.5
=      M0.1
AW>=   T37, 10
=      Q0.0
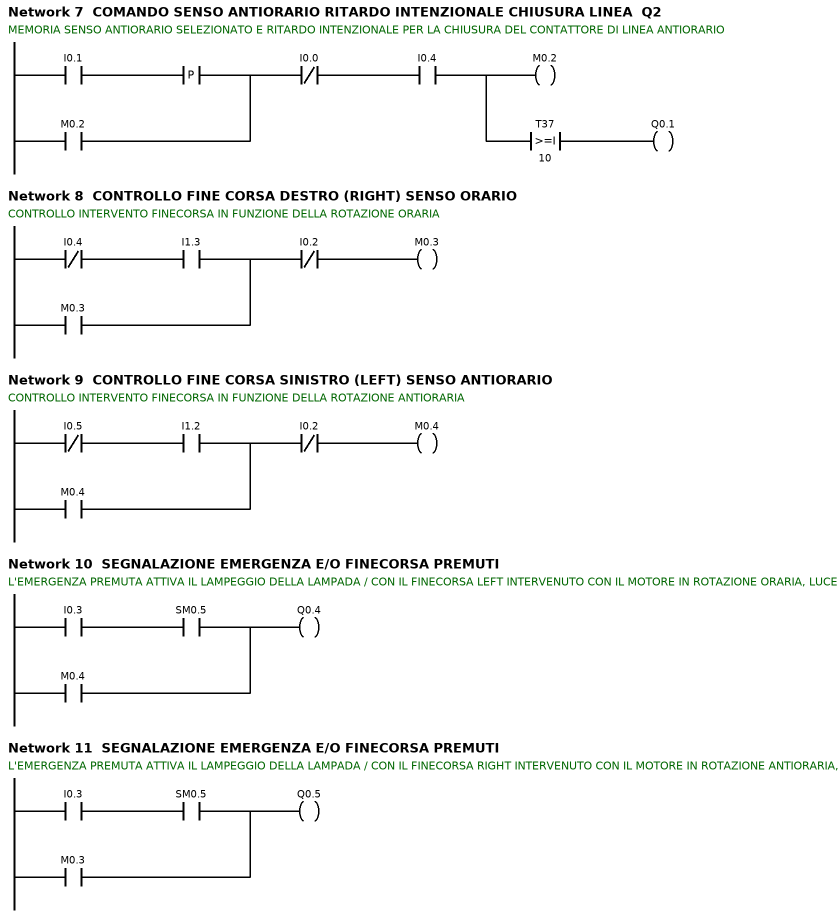
Network 7 // COMANDO SENSO ANTIORARIO RITARDO INTENZIONALE CHIUSURA LINEA  Q2
// MEMORIA SENSO ANTIORARIO SELEZIONATO E RITARDO INTENZIONALE PER LA CHIUSURA DEL CONTATTORE DI LINEA ANTIORARIO
LD     I0.1
EU
O      M0.2
AN     I0.0
A      I0.4
=      M0.2
AW>=   T37, 10
=      Q0.1
Network 8 // CONTROLLO FINE CORSA DESTRO (RIGHT) SENSO ORARIO
// CONTROLLO INTERVENTO FINECORSA IN FUNZIONE DELLA ROTAZIONE ORARIA
LDN    I0.4
A      I1.3
O      M0.3
AN     I0.2
=      M0.3
Network 9 // CONTROLLO FINE CORSA SINISTRO (LEFT) SENSO ANTIORARIO
// CONTROLLO INTERVENTO FINECORSA IN FUNZIONE DELLA ROTAZIONE ANTIORARIA
LDN    I0.5
A      I1.2
O      M0.4
AN     I0.2
=      M0.4
Network 10 // SEGNALAZIONE EMERGENZA E/O FINECORSA PREMUTI
// L'EMERGENZA PREMUTA ATTIVA IL LAMPEGGIO DELLA LAMPADA
// CON IL FINECORSA LEFT INTERVENUTO CON IL MOTORE IN ROTAZIONE ORARIA, LUCE FISSA
LD     I0.3
A      SM0.5
O      M0.4
=      Q0.4
Network 11 // SEGNALAZIONE EMERGENZA E/O FINECORSA PREMUTI
// L'EMERGENZA PREMUTA ATTIVA IL LAMPEGGIO DELLA LAMPADA
// CON IL FINECORSA RIGHT INTERVENUTO CON IL MOTORE IN ROTAZIONE ANTIORARIA, LUCE FISSA
LD     I0.3
A      SM0.5
O      M0.3
=      Q0.5
Network 12 // Titolo del segmento
// Commento del segmento
END_SUBROUTINE_BLOCK
